{attribute 'qualified_only'}
TYPE E_PFCA7_AcuumulationShutOff :
(
	ShutOffHasNotOccured := 0,
	ShutOffOccured	:= 1
);
END_TYPE

(* stored: Version 1.1.0.1, ProductVersion 3.1.4024.15
   DUT E_PFCA7_AcuumulationShutOff: Id {0be16eee-d552-02ea-2dc9-b7536dd9d7e2} *)
